SUBAPPLICATION AX_E_PERMIT_INVERT_1 (* Invertiertes Event-Freigabe-Gate mit Adapter-Signalen (AX_NOT_INIT + AX_E_PERMIT_1) *)
  (* Standard: 61499-2; Description: Copyright (c) 2026 Meisterschulen am Ostbahnhof This program and the accompanying materials are made available under the terms of the Eclipse Public License 2.0 which is available at https://www.eclipse.org/legal/epl-2.0/ SPDX-License-Identifier: EPL-2.0 *)
  (* Version 1.0, 2026-09-10, Franz Höpfinger, Meisterschulen am Ostbahnhof, initial implementation *)
  PACKAGE MyLib::sys;
  (* Documentation:
  Invertiertes Event-Freigabe-Gate (AX_NOT_INIT + AX_E_PERMIT_1)
   Kombination aus AX_NOT_INIT und AX_E_PERMIT_1 zur Freigabe von Ereignissen bei inaktiver (FALSE) Adapter-Bedingung.
   Funktionsbeschreibung
    - PERMIT (Socket AX): Eingehendes Freigabesignal.
   - AX_NOT_INIT: Invertiert das AX-Signal.
   - AX_E_PERMIT_1: Lässt Events von EI nach EO durch, wenn das invertierte Signal TRUE ist (also wenn PERMIT FALSE ist).
  *)
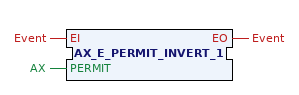
  EVENT_INPUT
    EI; (* Event input (wird durchgelassen wenn PERMIT FALSE ist) *)
  END_EVENT
  EVENT_OUTPUT
    EO; (* Event output (feuert wenn EI eintrifft und PERMIT FALSE ist) *)
  END_EVENT
  SOCKETS
    PERMIT : adapter::types::unidirectional::AX; (* Invertiertes Freigabesignal *)
  END_SOCKETS
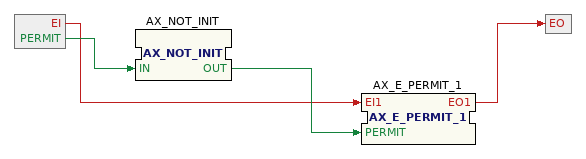
  FBS
    AX_NOT_INIT : adapter::booleanOperators::AX_NOT_INIT;
    AX_E_PERMIT_1 : adapter::events::unidirectional::AX_E_PERMIT_1;
  END_FBS
  EVENT_CONNECTIONS
    EI TO AX_E_PERMIT_1.EI1;
    AX_E_PERMIT_1.EO1 TO EO;
  END_CONNECTIONS
  ADAPTER_CONNECTIONS
    PERMIT TO AX_NOT_INIT.IN;
    AX_NOT_INIT.OUT TO AX_E_PERMIT_1.PERMIT;
  END_CONNECTIONS
END_SUBAPPLICATION
